FUNCTION_BLOCK Print
  (* Standard: 61499-2 *)
  (* Version 0.1, 2017-00-01, hpea485, UOA *)
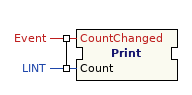
  EVENT_INPUT
    CountChanged WITH Count;
  END_EVENT
  VAR_INPUT
    Count : LINT;
  END_VAR
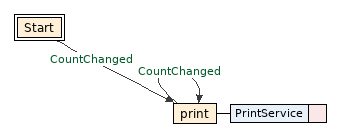
  EC_STATES
    Start;
    print : PrintService;
  END_STATES
  EC_TRANSITIONS
    Start TO print := CountChanged;
    print TO print := CountChanged;
  END_TRANSITIONS
  ALGORITHM PrintService IN C:
HEX = (unsigned int)me->Count; //printf("%lu\n", me->Count);
  END_ALGORITHM
END_FUNCTION_BLOCK
